(* IEC 61131-3 sources: uniset2/extensions/JScript/tools/st2js/tests/fixtures, 8 files *)

(* ---- fb_declaration.st ---- *)
FUNCTION_BLOCK MyController
VAR_INPUT
    SetPoint : REAL;
    Enable : BOOL;
END_VAR
VAR_OUTPUT
    Active : BOOL;
END_VAR
VAR
    counter : INT := 0;
END_VAR

counter := counter + 1;
IF SetPoint > 50.0 THEN
    Active := TRUE;
ELSE
    Active := FALSE;
END_IF;

END_FUNCTION_BLOCK

PROGRAM Main
VAR_INPUT
    Temperature : REAL;
END_VAR
VAR_OUTPUT
    Heater : BOOL;
END_VAR

Heater := TRUE;

END_PROGRAM

(* ---- control_flow.st ---- *)
PROGRAM ControlFlowTest
VAR
    x : INT := 0;
    i : INT;
    mystate : INT := 1;
    running : BOOL := TRUE;
END_VAR

CASE mystate OF
    1: x := 10;
    2: x := 20;
    3: x := 30;
ELSE
    x := 0;
END_CASE;

FOR i := 1 TO 10 BY 1 DO
    x := x + i;
END_FOR;

WHILE running DO
    x := x + 1;
END_WHILE;

REPEAT
    x := x - 1;
UNTIL x <= 0
END_REPEAT;

END_PROGRAM

(* ---- fb_calls.st ---- *)
PROGRAM Main
VAR_INPUT
    Enable : BOOL;
    Pulse : BOOL;
    ResetCmd : BOOL;
END_VAR
VAR_OUTPUT
    Output : BOOL;
    Count : INT;
END_VAR
VAR
    myTimer : TON;
    myCounter : CTU;
    myTrigger : R_TRIG;
    myLatch : RS;
END_VAR

myTimer(IN := Enable, PT := T#3000ms);
Output := myTimer.Q;

myCounter(CU := Pulse, RESET := ResetCmd, PV := 10);
Count := myCounter.CV;

myTrigger(CLK := Enable);

myLatch(SET := myTrigger.Q, RESET1 := ResetCmd);

END_PROGRAM

(* ---- minimal.st ---- *)
PROGRAM Main
VAR_INPUT
    Temperature : REAL;
    StartButton : BOOL;
END_VAR
VAR_OUTPUT
    Heater : BOOL;
    Alarm : BOOL;
END_VAR
VAR
    state : INT := 0;
END_VAR

IF StartButton THEN
    Heater := TRUE;
END_IF;

IF Temperature > 80.0 THEN
    Alarm := TRUE;
END_IF;

END_PROGRAM

(* ---- multi_program.st ---- *)
PROGRAM Alarms
VAR
    alarmActive : BOOL := FALSE;
    alarmTimer : TON;
END_VAR

alarmTimer(IN := alarmActive, PT := T#10s);
IF alarmTimer.Q THEN
    alarmActive := FALSE;
END_IF;

END_PROGRAM

PROGRAM HMI_Update
VAR
    counter : INT := 0;
END_VAR

counter := counter + 1;

END_PROGRAM

PROGRAM Main
VAR_INPUT
    Temperature : REAL;
    Enable : BOOL;
END_VAR
VAR_OUTPUT
    Heater : BOOL;
END_VAR
VAR
    state : INT := 0;
END_VAR

IF Enable THEN
    state := 1;
END_IF;

IF state = 1 THEN
    IF Temperature < 20.0 THEN
        Heater := TRUE;
    ELSE
        Heater := FALSE;
    END_IF;
END_IF;

Alarms();
HMI_Update();

END_PROGRAM

(* ---- scale_test.st ---- *)
PROGRAM ScaleTest
VAR_INPUT
    Temperature : REAL;
    Pressure : REAL;
    StartButton : BOOL;
END_VAR
VAR_OUTPUT
    ValvePos : REAL;
    Alarm : BOOL;
END_VAR
VAR
    setpoint : REAL := 50.0;
END_VAR

IF Temperature > setpoint THEN
    ValvePos := Temperature - setpoint;
    Alarm := TRUE;
END_IF;

END_PROGRAM

(* ---- struct_array.st ---- *)
TYPE SensorData :
STRUCT
    value : INT;
    scale : REAL := 1.0;
    valid : BOOL;
END_STRUCT
END_TYPE

PROGRAM StructArrayTest
VAR
    sensor : SensorData;
    readings : ARRAY[1..5] OF INT;
    name : STRING := 'test';
    timeout : TIME := T#5s;
END_VAR

sensor.value := 42;
sensor.valid := TRUE;
readings[1] := sensor.value;
readings[3] := 100;

END_PROGRAM

(* ---- thermostat.st ---- *)
TYPE TempConfig :
STRUCT
    setpoint : REAL := 20.0;
    hysteresis : REAL := 2.0;
    maxTemp : REAL := 95.0;
END_STRUCT
END_TYPE

PROGRAM Thermostat
VAR_INPUT
    CurrentTemp : REAL;
    Enable : BOOL;
    Reset : BOOL;
END_VAR
VAR_OUTPUT
    HeaterOn : BOOL;
    AlarmHigh : BOOL;
    CycleCount : INT;
END_VAR
VAR
    config : TempConfig;
    onDelay : TON;
    offDelay : TOF;
    startEdge : R_TRIG;
    cycleCounter : CTU;
    state : INT := 0;
    i : INT;
END_VAR

startEdge(CLK := Enable);
IF startEdge.Q THEN
    state := 1;
END_IF;

CASE state OF
    0: (* Idle *)
        HeaterOn := FALSE;
    1: (* Running *)
        IF CurrentTemp < config.setpoint - config.hysteresis THEN
            HeaterOn := TRUE;
        ELSIF CurrentTemp > config.setpoint + config.hysteresis THEN
            HeaterOn := FALSE;
        END_IF;

        onDelay(IN := HeaterOn, PT := T#5s);
        cycleCounter(CU := onDelay.Q, RESET := Reset, PV := 100);
        CycleCount := cycleCounter.CV;
    2: (* Alarm *)
        HeaterOn := FALSE;
END_CASE;

IF CurrentTemp > config.maxTemp THEN
    AlarmHigh := TRUE;
    state := 2;
END_IF;

IF Reset THEN
    state := 0;
    AlarmHigh := FALSE;
END_IF;

END_PROGRAM
